FUNCTION_BLOCK StringBuilderExtBufferTest EXTENDS TcUnit.FB_TestSuite
VAR
END_VAR

AppendAndClear();

METHOD AppendAndClear : BOOL
VAR
	buffer : STRING(2000);
	builder : StringBuilderExtBuffer := (Buffer := ToAnyType(buffer));
	
	testValue : STRING := ' very long strings';
END_VAR
TcUnit.TEST('Append and Clear');

builder
	.Clear()
	.Append('SB with external buffer')
	.Append(' is meant for')
	.AppendByPointer(ADR(testValue));

AssertEquals_STRING(
	Expected := 'SB with external buffer is meant for very long strings',
	Actual := buffer,
	Message := 'Strings should be properly appended');

builder.Clear();

AssertEquals_BOOL(
	Expected := TRUE,
	Actual := builder.IsEmpty,
	Message := 'Buffer should be empty');
	
TEST_FINISHED();
END_METHOD

END_FUNCTION_BLOCK

(* stored: Version 1.1.0.1, ProductVersion 3.1.4024.15
   POU StringBuilderExtBufferTest: Id {c33f3568-737d-0f8d-016e-c400b31ebd8d}, SpecialFunc None
   Method AppendAndClear: Id {456e8ba9-e0db-0c67-100d-b68bbdeccdd7} *)
